{attribute 'qualified_only'}
{attribute 'strict'}
{attribute 'to_string'}
TYPE ST110_Cylinders_e :
(
    VakuumgreiferLinks,
    VakuumgreiferRechts,
    _max
);
END_TYPE

(* stored: Version 1.1.0.1, ProductVersion 3.1.4024.6
   EnumerationTextList ST110_Cylinders_e: Id {74b7fae7-3f3b-454e-8d05-e84f34a46845} *)
